Staubli VAL3: StartMotion.pgx

public program StartMotion(string x_sPath)
begin
  //
  taskCreate "motion",100,SingleMotion(x_sPath,true,0)
  wait(taskStatus("motion")==1)
end
